// TwinCAT 3 PLC project
// project tree:
//   POUs/ func_f1.TcPOU, func_f2.TcPOU, func_f3.TcPOU, makeTupleStruct_1.TcPOU, proj0_TupleStruct_1.TcPOU (not stored), proj1_TupleStruct_1.TcPOU (not stored), MAIN.TcPOU
//   DUTs/ STATE.TcDUT, TupleStruct_1.TcDUT (not stored)
//   GVLs/ INPUTS.TcGVL, TIMERS.TcGVL (not stored)

// ---- DUTs/STATE.TcDUT
TYPE STATE:
    STRUCT
        curTime: LREAL;
        dvar_M_aut_x AT %Q*: DINT;
        dvar_M_aut_y AT %Q*: DINT;
        dvar_M_aut_z AT %Q*: DINT;
    END_STRUCT
END_TYPE

// ---- GVLs/INPUTS.TcGVL

      VAR_GLOBAL // INPUTS
    ivar_i AT %I*: DINT;
END_VAR

// ---- POUs/func_f1.TcPOU
FUNCTION func_f1: DINT
VAR_INPUT
    farg2_f1_x: DINT;
END_VAR
VAR
    farg_f1_x: DINT;
END_VAR

farg_f1_x := farg2_f1_x;
IF ((farg_f1_x) <= (0)) THEN
    func_f1 := farg_f1_x;
    RETURN;
END_IF;
farg_f1_x := (farg_f1_x) + (1);
func_f1 := func_f2(farg_f1_x);
RETURN;

END_FUNCTION

// ---- POUs/func_f2.TcPOU
FUNCTION func_f2: DINT
VAR_INPUT
    farg2_f2_x: DINT;
END_VAR
VAR
    farg_f2_x: DINT;
END_VAR

farg_f2_x := farg2_f2_x;
IF ((farg_f2_x) <= (0)) THEN
    func_f2 := farg_f2_x;
    RETURN;
END_IF;
farg_f2_x := (farg_f2_x) - (2);
func_f2 := func_f1(farg_f2_x);
RETURN;

END_FUNCTION

// ---- POUs/func_f3.TcPOU
FUNCTION func_f3: DINT
VAR_INPUT
    farg_f3_z: DINT;
END_VAR
VAR
    fvar_f3_x: DINT;
    fvar_f3_y: DINT;
    tmp0: DINT;
    tmp1: DINT;
END_VAR

// Initialize local variables.
fvar_f3_x := 1;
fvar_f3_y := 2;

// Actual function body.
tmp0 := fvar_f3_x;
tmp1 := fvar_f3_y;
tmp0 := proj0_TupleStruct_1(makeTupleStruct_1(fvar_f3_y, fvar_f3_x));
tmp1 := proj1_TupleStruct_1(makeTupleStruct_1(fvar_f3_y, fvar_f3_x));
fvar_f3_x := tmp0;
fvar_f3_y := tmp1;
func_f3 := ((fvar_f3_x) + (fvar_f3_y)) + (farg_f3_z);
RETURN;

END_FUNCTION

// ---- POUs/makeTupleStruct_1.TcPOU
FUNCTION makeTupleStruct_1: TupleStruct_1
VAR_INPUT
    field0: DINT;
    field1: DINT;
END_VAR
VAR
    rslt: TupleStruct_1;
END_VAR

rslt.field0 := field0;
rslt.field1 := field1;
makeTupleStruct_1 := rslt;

END_FUNCTION

// ---- POUs/MAIN.TcPOU
PROGRAM MAIN
VAR_OUTPUT
    timerValue0: TIME;
    timerValue1: TIME;
END_VAR
VAR
    cnt: LINT;
    first: BOOL := TRUE;
    curTimerValue: TIME;
    state0: STATE;
    curTime: LREAL;
    loopsKilled: LINT;
END_VAR
VAR_TEMP
    lastTimerValue: TIME;
    curDeltaTime: TIME;
    curDeltaSecs: LREAL;
    state1: STATE;
    progress: BOOL;
    loopCount: INT;
END_VAR


// Handle 'time' and cycle time.
cnt := cnt + 1;

timer0(IN := curTimer = 0, PT := T#1D);
timer1(IN := curTimer = 1, PT := T#1D);
timerValue0 := timer0.ET;
timerValue1 := timer1.ET;

lastTimerValue := curTimerValue;
IF curTimer = 0 THEN
    curTimerValue := timerValue0;
ELSE
    curTimerValue := timerValue1;
END_IF;
curDeltaTime := curTimerValue - lastTimerValue;
curDeltaSecs := TIME_TO_LREAL(curDeltaTime) / 1000;
curTime := curTime + curDeltaSecs;

IF cnt MOD 10 = 0 THEN
    curTimer := 1 - curTimer;
    curTimerValue := T#0S;
    timer0(IN := curTimer = 0, PT := T#1D);
    timer1(IN := curTimer = 1, PT := T#1D);
    timerValue0 := timer0.ET;
    timerValue1 := timer1.ET;
END_IF;

IF first THEN
    first := FALSE;

    // Initialize state variables for initial state.
    state0.dvar_M_aut_x := 10;
    state0.dvar_M_aut_y := func_f1(10);
    state0.dvar_M_aut_z := func_f3(0);
ELSE
    // Update continuous variables for time delay.

    state0.curTime := curTime;
END_IF;

// Event loop.
WHILE TRUE DO
    progress := FALSE;

    // Event "tau".
    IF NOT progress THEN
        IF (state0.dvar_M_aut_y) = (0) THEN
            progress := TRUE;
            state1 := state0;

            state1.dvar_M_aut_y := (ivar_i) + (state0.dvar_M_aut_z);

            state0 := state1;
        END_IF;
    END_IF;

    // Done with events?
    IF NOT progress THEN
        EXIT;
    END_IF;

    // Protect against events that are always enabled.
    loopCount := loopCount + 1;
    IF loopCount >= 100 THEN
        loopsKilled := loopsKilled + 1;
        EXIT;
    END_IF;
END_WHILE;

END_PROGRAM
